PROGRAM RC4_CRYPT_DEMO
VAR
	RC4_CRYPT_STREAM: RC4_CRYPT_STREAM;
	(* buf : ARRAY [0..63] OF BYTE := 107,117,114,116;*) (* kurt *)
	buf : ARRAY [0..63] OF BYTE := 110,60,3,219; (* crypt *)
	mode: INT;
	key: STRING := '1234';
	size: UDINT := 4;
	pos: UDINT;
END_VAR

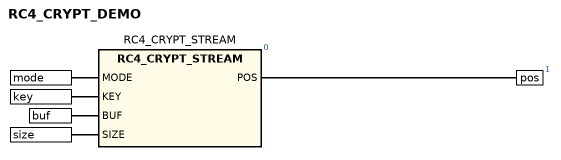
RC4_CRYPT_STREAM(MODE := mode, KEY := key, BUF := buf, SIZE := size);
pos := RC4_CRYPT_STREAM.POS;

END_PROGRAM

(* stored: Version 1.1.0.1, ProductVersion 3.1.4022.7
   POU RC4_CRYPT_DEMO: Id {9e200141-1308-4b30-9302-fd1dbb9246fb}, SpecialFunc None *)
